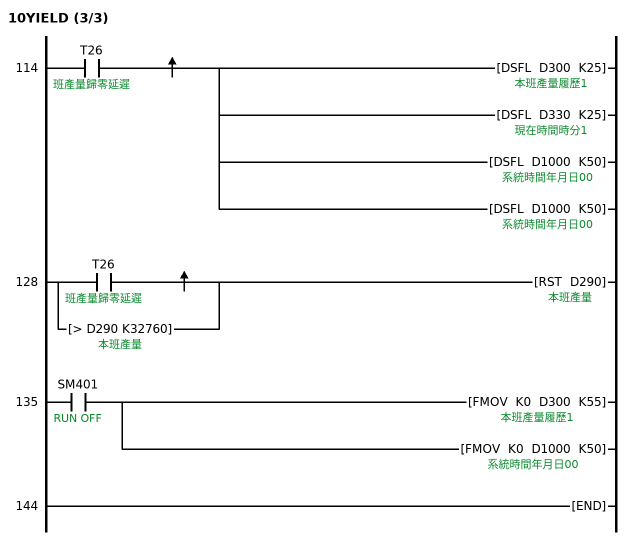
[picture p48: ladder of 10YIELD, rungs at steps 114 to 144]
114   LD      T26  ; 班產量歸零延遲
      MEP
      DSFL    D300 K25
      DSFL    D330 K25
      DSFL    D1000 K50
      DSFL    D1000 K50
128   LD      T26  ; 班產量歸零延遲
      MEP
      OR>     D290 K32760  ; 本班產量
      RST     D290  ; 本班產量
135   LD      SM401  ; RUN OFF
      FMOV    K0 D300 K55
      FMOV    K0 D1000 K50
144   END
END_PROGRAM

PROGRAM 11MAINTE
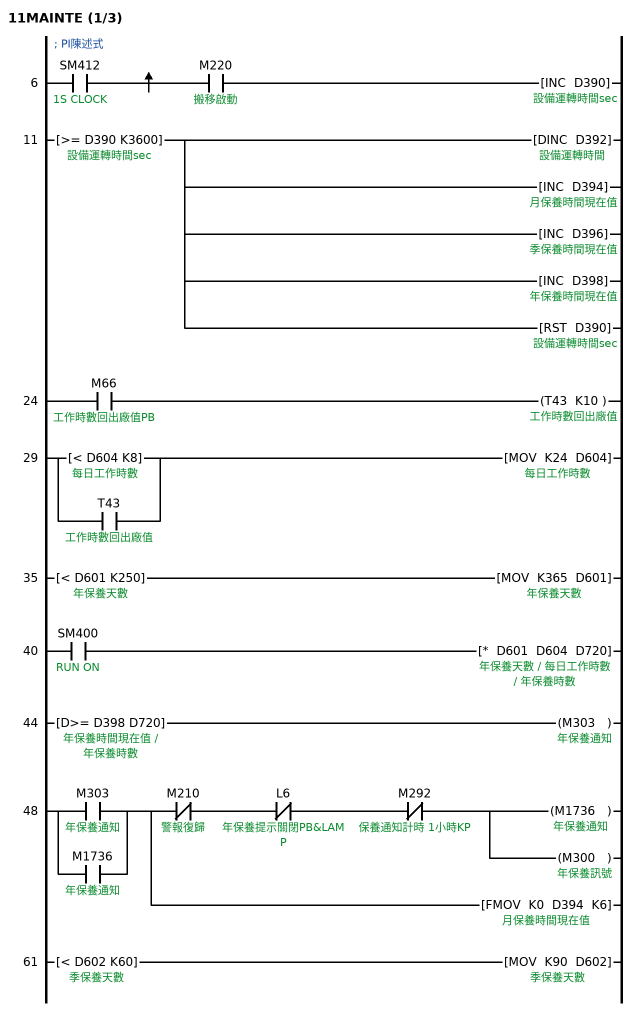
; PI陳述式
6     LD      SM412  ; 1S CLOCK
      MEP
      AND     M220  ; 搬移啟動
      INC     D390  ; 設備運轉時間sec
11    LD>=    D390 K3600  ; 設備運轉時間sec
      DINC    D392  ; 設備運轉時間
      INC     D394  ; 月保養時間現在值
      INC     D396  ; 季保養時間現在值
      INC     D398  ; 年保養時間現在值
      RST     D390  ; 設備運轉時間sec
24    LD      M66  ; 工作時數回出廠值PB
      OUT     T43 K10  ; 工作時數回出廠值
29    LD<     D604 K8  ; 每日工作時數
      OR      T43  ; 工作時數回出廠值
      MOV     K24 D604
35    LD<     D601 K250  ; 年保養天數
      MOV     K365 D601
40    LD      SM400  ; RUN ON
      *       D601 D604 D720  ; 年保養時數
44    LDD>=   D398 D720  ; 年保養時間現在值 / 年保養時數
      OUT     M303  ; 年保養通知
48    LD      M303  ; 年保養通知
      OR      M1736  ; 年保養通知
      MPS
      ANI     M210  ; 警報復歸
      ANI     L6  ; 年保養提示關閉PB&LAMP
      ANI     M292  ; 保養通知計時 1小時KP
      OUT     M1736  ; 年保養通知
      OUT     M300  ; 年保養訊號
      MPP
      FMOV    K0 D394 K6
61    LD<     D602 K60  ; 季保養天數
      MOV     K90 D602
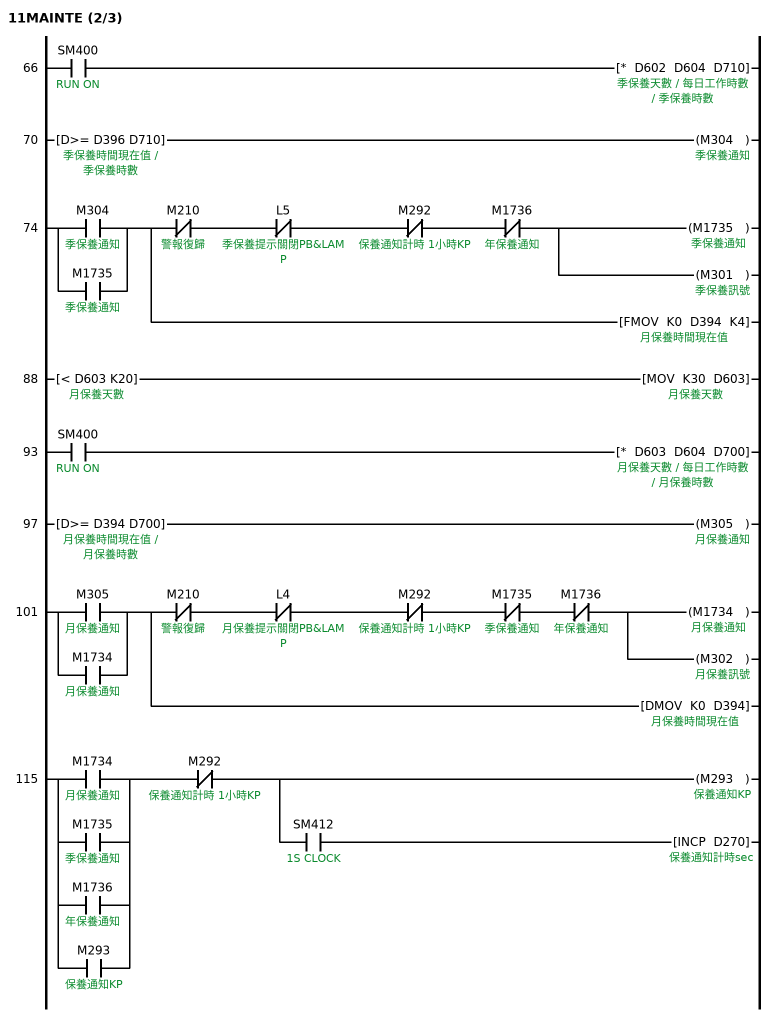
66    LD      SM400  ; RUN ON
      *       D602 D604 D710  ; 季保養時數
70    LDD>=   D396 D710  ; 季保養時間現在值 / 季保養時數
      OUT     M304  ; 季保養通知
74    LD      M304  ; 季保養通知
      OR      M1735  ; 季保養通知
      MPS
      ANI     M210  ; 警報復歸
      ANI     L5  ; 季保養提示關閉PB&LAMP
      ANI     M292  ; 保養通知計時 1小時KP
      ANI     M1736  ; 年保養通知
      OUT     M1735  ; 季保養通知
      OUT     M301  ; 季保養訊號
      MPP
      FMOV    K0 D394 K4
88    LD<     D603 K20  ; 月保養天數
      MOV     K30 D603
93    LD      SM400  ; RUN ON
      *       D603 D604 D700  ; 月保養時數
97    LDD>=   D394 D700  ; 月保養時間現在值 / 月保養時數
      OUT     M305  ; 月保養通知
101   LD      M305  ; 月保養通知
      OR      M1734  ; 月保養通知
      MPS
      ANI     M210  ; 警報復歸
      ANI     L4  ; 月保養提示關閉PB&LAMP
      ANI     M292  ; 保養通知計時 1小時KP
      ANI     M1735  ; 季保養通知
      ANI     M1736  ; 年保養通知
      OUT     M1734  ; 月保養通知
      OUT     M302  ; 月保養訊號
      MPP
      DMOV    K0 D394
115   LD      M1734  ; 月保養通知
      OR      M1735  ; 季保養通知
      OR      M1736  ; 年保養通知
      OR      M293  ; 保養通知KP
      ANI     M292  ; 保養通知計時 1小時KP
      OUT     M293  ; 保養通知KP
      AND     SM412  ; 1S CLOCK
      INCP    D270  ; 保養通知計時sec
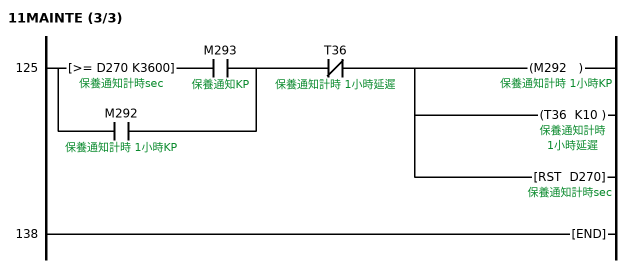
125   LD>=    D270 K3600  ; 保養通知計時sec
      AND     M293  ; 保養通知KP
      OR      M292  ; 保養通知計時 1小時KP
      ANI     T36  ; 保養通知計時 1小時延遲
      OUT     M292  ; 保養通知計時 1小時KP
      OUT     T36 K10  ; 保養通知計時 1小時延遲
      RST     D270  ; 保養通知計時sec
138   END
END_PROGRAM

PROGRAM 12ALARM1
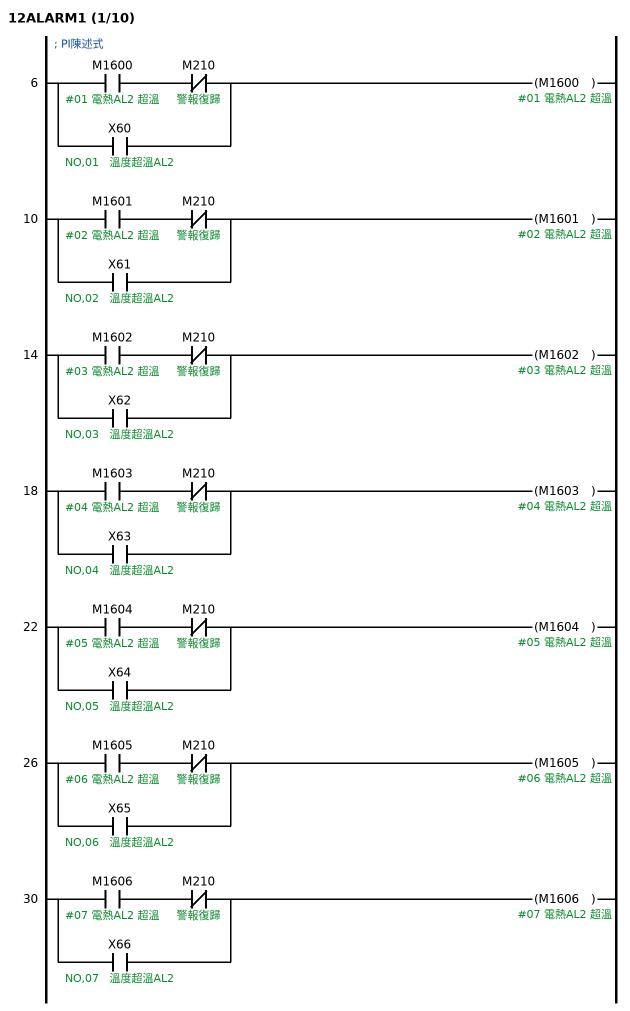
; PI陳述式
6     LD      M1600  ; #01 電熱AL2 超溫
      ANI     M210  ; 警報復歸
      OR      X60  ; NO,01   溫度超溫AL2
      OUT     M1600  ; #01 電熱AL2 超溫
10    LD      M1601  ; #02 電熱AL2 超溫
      ANI     M210  ; 警報復歸
      OR      X61  ; NO,02   溫度超溫AL2
      OUT     M1601  ; #02 電熱AL2 超溫
14    LD      M1602  ; #03 電熱AL2 超溫
      ANI     M210  ; 警報復歸
      OR      X62  ; NO,03   溫度超溫AL2
      OUT     M1602  ; #03 電熱AL2 超溫
18    LD      M1603  ; #04 電熱AL2 超溫
      ANI     M210  ; 警報復歸
      OR      X63  ; NO,04   溫度超溫AL2
      OUT     M1603  ; #04 電熱AL2 超溫
22    LD      M1604  ; #05 電熱AL2 超溫
      ANI     M210  ; 警報復歸
      OR      X64  ; NO,05   溫度超溫AL2
      OUT     M1604  ; #05 電熱AL2 超溫
26    LD      M1605  ; #06 電熱AL2 超溫
      ANI     M210  ; 警報復歸
      OR      X65  ; NO,06   溫度超溫AL2
      OUT     M1605  ; #06 電熱AL2 超溫
30    LD      M1606  ; #07 電熱AL2 超溫
      ANI     M210  ; 警報復歸
      OR      X66  ; NO,07   溫度超溫AL2
      OUT     M1606  ; #07 電熱AL2 超溫
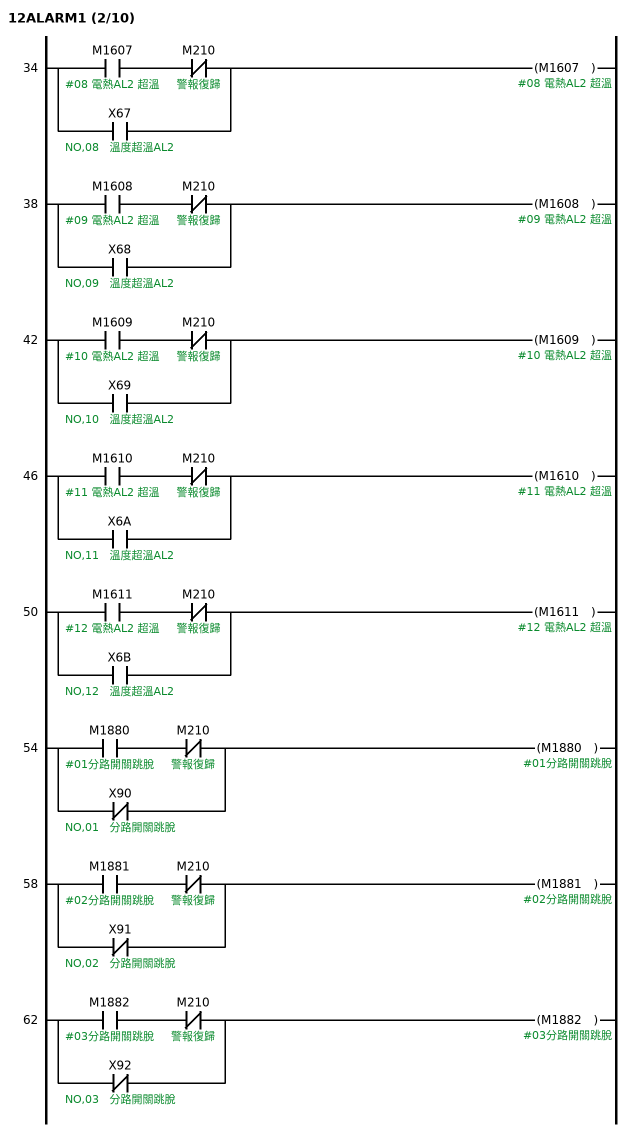
34    LD      M1607  ; #08 電熱AL2 超溫
      ANI     M210  ; 警報復歸
      OR      X67  ; NO,08   溫度超溫AL2
      OUT     M1607  ; #08 電熱AL2 超溫
38    LD      M1608  ; #09 電熱AL2 超溫
      ANI     M210  ; 警報復歸
      OR      X68  ; NO,09   溫度超溫AL2
      OUT     M1608  ; #09 電熱AL2 超溫
42    LD      M1609  ; #10 電熱AL2 超溫
      ANI     M210  ; 警報復歸
      OR      X69  ; NO,10   溫度超溫AL2
      OUT     M1609  ; #10 電熱AL2 超溫
46    LD      M1610  ; #11 電熱AL2 超溫
      ANI     M210  ; 警報復歸
      OR      X6A  ; NO,11   溫度超溫AL2
      OUT     M1610  ; #11 電熱AL2 超溫
50    LD      M1611  ; #12 電熱AL2 超溫
      ANI     M210  ; 警報復歸
      OR      X6B  ; NO,12   溫度超溫AL2
      OUT     M1611  ; #12 電熱AL2 超溫
54    LD      M1880  ; #01分路開關跳脫
      ANI     M210  ; 警報復歸
      ORI     X90  ; NO,01   分路開關跳脫
      OUT     M1880  ; #01分路開關跳脫
58    LD      M1881  ; #02分路開關跳脫
      ANI     M210  ; 警報復歸
      ORI     X91  ; NO,02   分路開關跳脫
      OUT     M1881  ; #02分路開關跳脫
62    LD      M1882  ; #03分路開關跳脫
      ANI     M210  ; 警報復歸
      ORI     X92  ; NO,03   分路開關跳脫
      OUT     M1882  ; #03分路開關跳脫
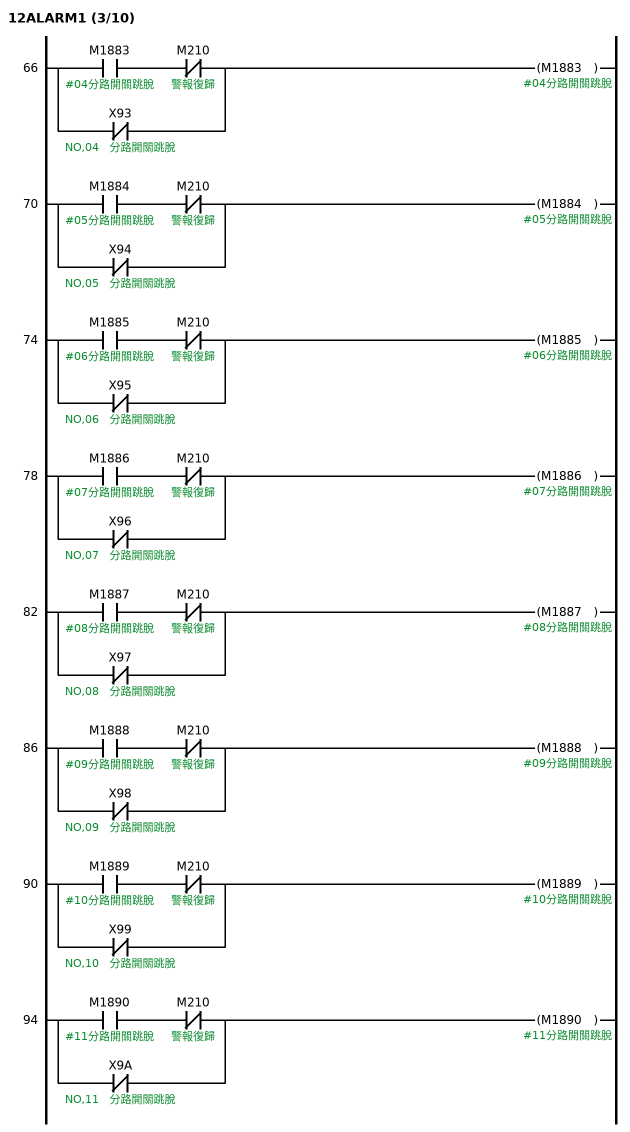
66    LD      M1883  ; #04分路開關跳脫
      ANI     M210  ; 警報復歸
      ORI     X93  ; NO,04   分路開關跳脫
      OUT     M1883  ; #04分路開關跳脫
70    LD      M1884  ; #05分路開關跳脫
      ANI     M210  ; 警報復歸
      ORI     X94  ; NO,05   分路開關跳脫
      OUT     M1884  ; #05分路開關跳脫
74    LD      M1885  ; #06分路開關跳脫
      ANI     M210  ; 警報復歸
      ORI     X95  ; NO,06   分路開關跳脫
      OUT     M1885  ; #06分路開關跳脫
78    LD      M1886  ; #07分路開關跳脫
      ANI     M210  ; 警報復歸
      ORI     X96  ; NO,07   分路開關跳脫
      OUT     M1886  ; #07分路開關跳脫
82    LD      M1887  ; #08分路開關跳脫
      ANI     M210  ; 警報復歸
      ORI     X97  ; NO,08   分路開關跳脫
      OUT     M1887  ; #08分路開關跳脫
86    LD      M1888  ; #09分路開關跳脫
      ANI     M210  ; 警報復歸
      ORI     X98  ; NO,09   分路開關跳脫
      OUT     M1888  ; #09分路開關跳脫
90    LD      M1889  ; #10分路開關跳脫
      ANI     M210  ; 警報復歸
      ORI     X99  ; NO,10   分路開關跳脫
      OUT     M1889  ; #10分路開關跳脫
94    LD      M1890  ; #11分路開關跳脫
      ANI     M210  ; 警報復歸
      ORI     X9A  ; NO,11   分路開關跳脫
      OUT     M1890  ; #11分路開關跳脫
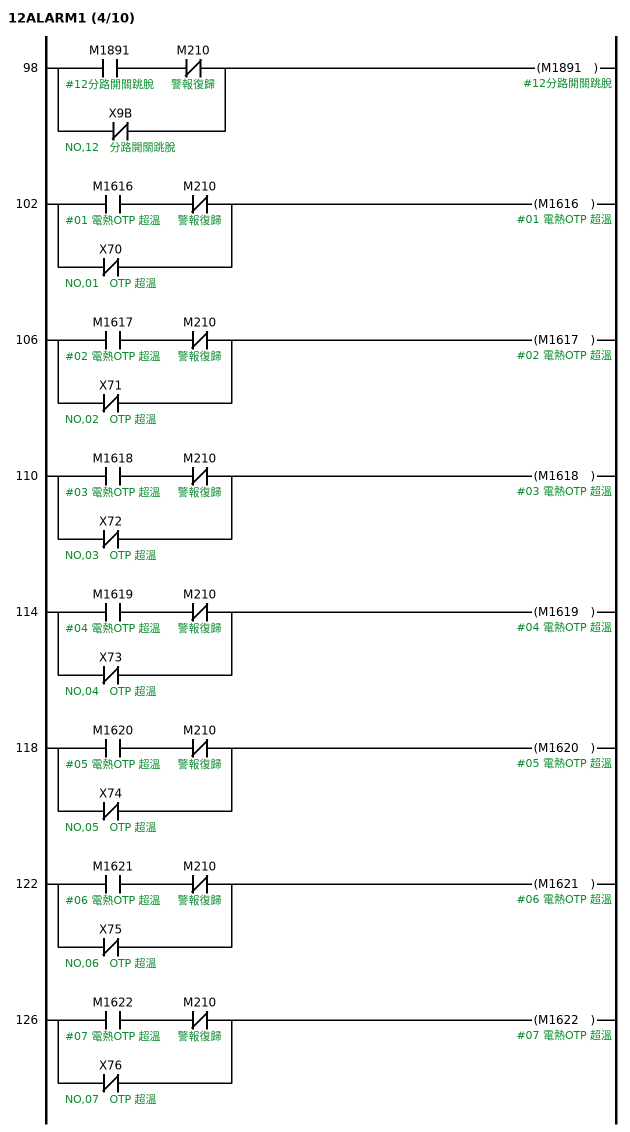
98    LD      M1891  ; #12分路開關跳脫
      ANI     M210  ; 警報復歸
      ORI     X9B  ; NO,12   分路開關跳脫
      OUT     M1891  ; #12分路開關跳脫
102   LD      M1616  ; #01 電熱OTP 超溫
      ANI     M210  ; 警報復歸
      ORI     X70  ; NO,01   OTP 超溫
      OUT     M1616  ; #01 電熱OTP 超溫
106   LD      M1617  ; #02 電熱OTP 超溫
      ANI     M210  ; 警報復歸
      ORI     X71  ; NO,02   OTP 超溫
      OUT     M1617  ; #02 電熱OTP 超溫
110   LD      M1618  ; #03 電熱OTP 超溫
      ANI     M210  ; 警報復歸
      ORI     X72  ; NO,03   OTP 超溫
      OUT     M1618  ; #03 電熱OTP 超溫
114   LD      M1619  ; #04 電熱OTP 超溫
      ANI     M210  ; 警報復歸
      ORI     X73  ; NO,04   OTP 超溫
      OUT     M1619  ; #04 電熱OTP 超溫
118   LD      M1620  ; #05 電熱OTP 超溫
      ANI     M210  ; 警報復歸
      ORI     X74  ; NO,05   OTP 超溫
      OUT     M1620  ; #05 電熱OTP 超溫
122   LD      M1621  ; #06 電熱OTP 超溫
      ANI     M210  ; 警報復歸
      ORI     X75  ; NO,06   OTP 超溫
      OUT     M1621  ; #06 電熱OTP 超溫
126   LD      M1622  ; #07 電熱OTP 超溫
      ANI     M210  ; 警報復歸
      ORI     X76  ; NO,07   OTP 超溫
      OUT     M1622  ; #07 電熱OTP 超溫
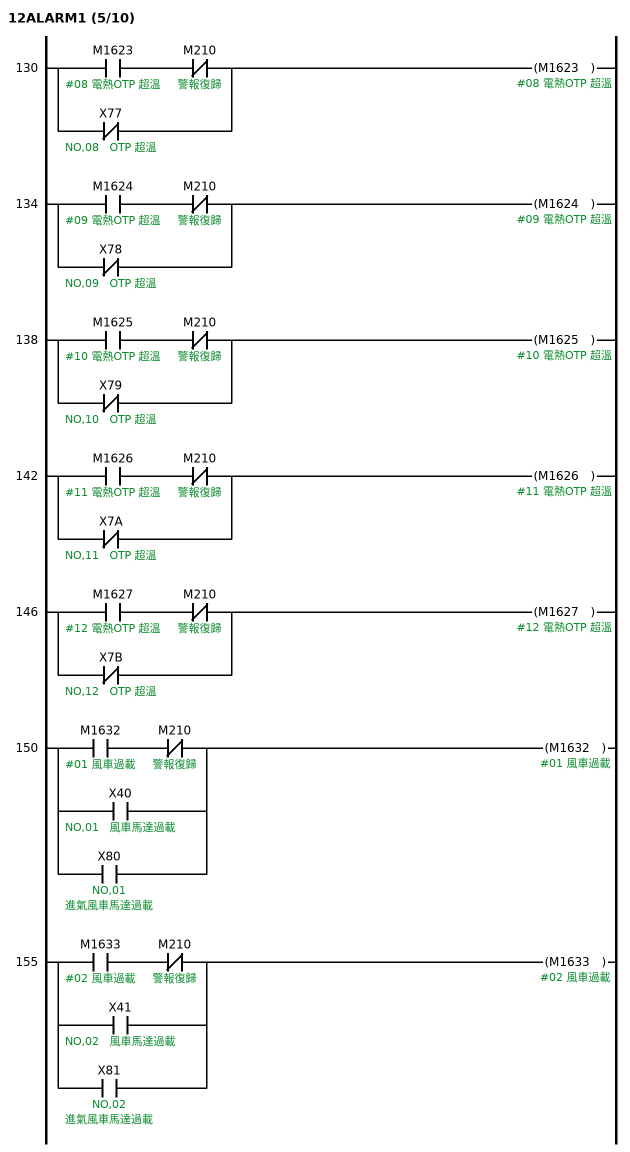
130   LD      M1623  ; #08 電熱OTP 超溫
      ANI     M210  ; 警報復歸
      ORI     X77  ; NO,08   OTP 超溫
      OUT     M1623  ; #08 電熱OTP 超溫
134   LD      M1624  ; #09 電熱OTP 超溫
      ANI     M210  ; 警報復歸
      ORI     X78  ; NO,09   OTP 超溫
      OUT     M1624  ; #09 電熱OTP 超溫
138   LD      M1625  ; #10 電熱OTP 超溫
      ANI     M210  ; 警報復歸
      ORI     X79  ; NO,10   OTP 超溫
      OUT     M1625  ; #10 電熱OTP 超溫
142   LD      M1626  ; #11 電熱OTP 超溫
      ANI     M210  ; 警報復歸
      ORI     X7A  ; NO,11   OTP 超溫
      OUT     M1626  ; #11 電熱OTP 超溫
146   LD      M1627  ; #12 電熱OTP 超溫
      ANI     M210  ; 警報復歸
      ORI     X7B  ; NO,12   OTP 超溫
      OUT     M1627  ; #12 電熱OTP 超溫
150   LD      M1632  ; #01 風車過載
      ANI     M210  ; 警報復歸
      OR      X40  ; NO,01   風車馬達過載
      OR      X80  ; NO,01   進氣風車馬達過載
      OUT     M1632  ; #01 風車過載
155   LD      M1633  ; #02 風車過載
      ANI     M210  ; 警報復歸
      OR      X41  ; NO,02   風車馬達過載
      OR      X81  ; NO,02   進氣風車馬達過載
      OUT     M1633  ; #02 風車過載
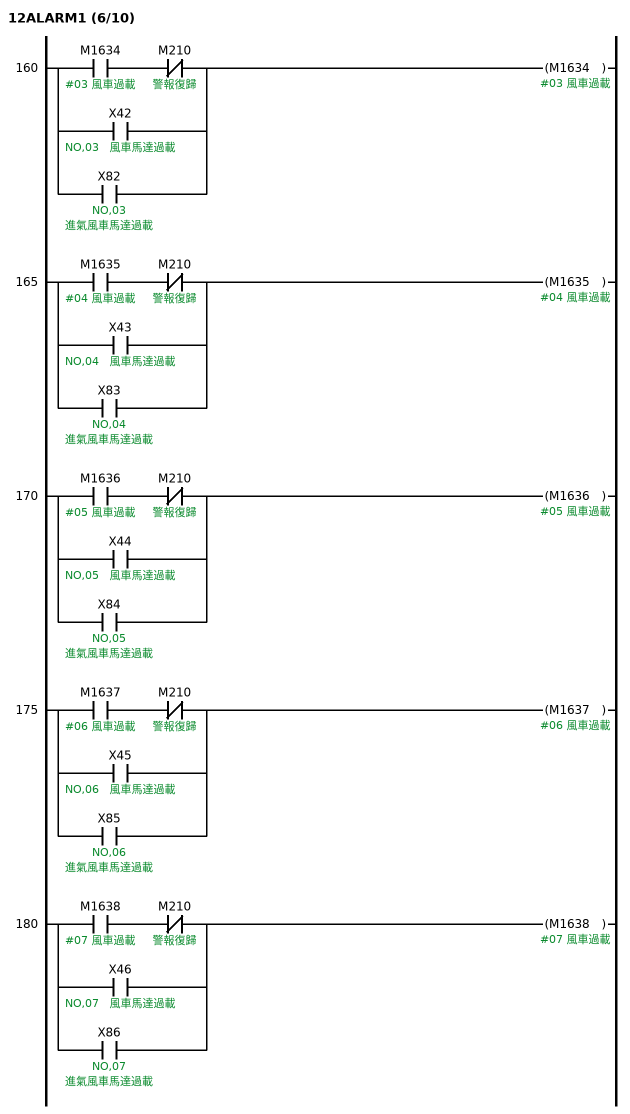
160   LD      M1634  ; #03 風車過載
      ANI     M210  ; 警報復歸
      OR      X42  ; NO,03   風車馬達過載
      OR      X82  ; NO,03   進氣風車馬達過載
      OUT     M1634  ; #03 風車過載
165   LD      M1635  ; #04 風車過載
      ANI     M210  ; 警報復歸
      OR      X43  ; NO,04   風車馬達過載
      OR      X83  ; NO,04   進氣風車馬達過載
      OUT     M1635  ; #04 風車過載
170   LD      M1636  ; #05 風車過載
      ANI     M210  ; 警報復歸
      OR      X44  ; NO,05   風車馬達過載
      OR      X84  ; NO,05   進氣風車馬達過載
      OUT     M1636  ; #05 風車過載
175   LD      M1637  ; #06 風車過載
      ANI     M210  ; 警報復歸
      OR      X45  ; NO,06   風車馬達過載
      OR      X85  ; NO,06   進氣風車馬達過載
      OUT     M1637  ; #06 風車過載
180   LD      M1638  ; #07 風車過載
      ANI     M210  ; 警報復歸
      OR      X46  ; NO,07   風車馬達過載
      OR      X86  ; NO,07   進氣風車馬達過載
      OUT     M1638  ; #07 風車過載
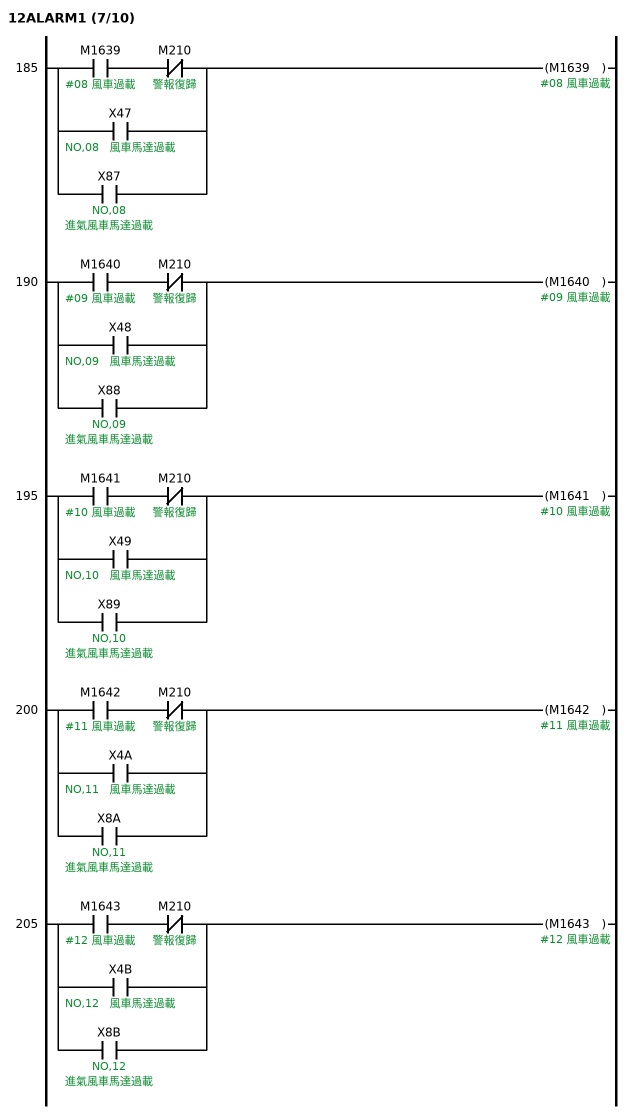
185   LD      M1639  ; #08 風車過載
      ANI     M210  ; 警報復歸
      OR      X47  ; NO,08   風車馬達過載
      OR      X87  ; NO,08   進氣風車馬達過載
      OUT     M1639  ; #08 風車過載
190   LD      M1640  ; #09 風車過載
      ANI     M210  ; 警報復歸
      OR      X48  ; NO,09   風車馬達過載
      OR      X88  ; NO,09   進氣風車馬達過載
      OUT     M1640  ; #09 風車過載
195   LD      M1641  ; #10 風車過載
      ANI     M210  ; 警報復歸
      OR      X49  ; NO,10   風車馬達過載
      OR      X89  ; NO,10   進氣風車馬達過載
      OUT     M1641  ; #10 風車過載
200   LD      M1642  ; #11 風車過載
      ANI     M210  ; 警報復歸
      OR      X4A  ; NO,11   風車馬達過載
      OR      X8A  ; NO,11   進氣風車馬達過載
      OUT     M1642  ; #11 風車過載
205   LD      M1643  ; #12 風車過載
      ANI     M210  ; 警報復歸
      OR      X4B  ; NO,12   風車馬達過載
      OR      X8B  ; NO,12   進氣風車馬達過載
      OUT     M1643  ; #12 風車過載
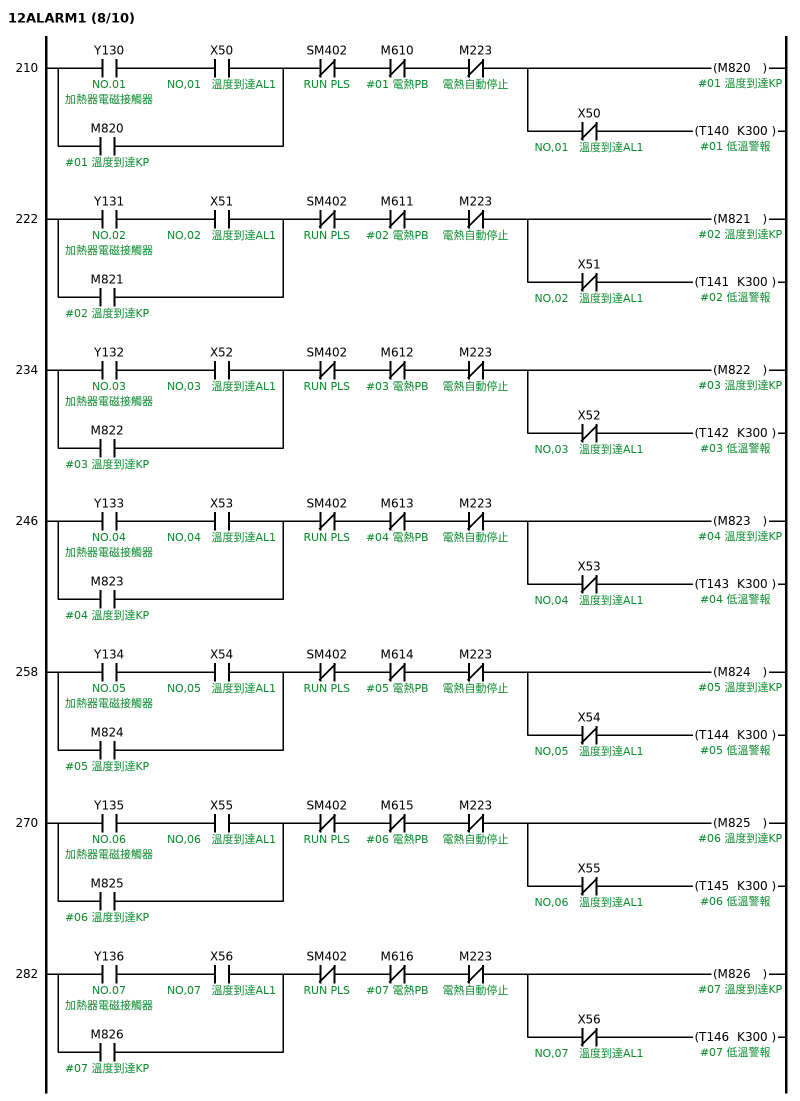
210   LD      Y130  ; NO.01   加熱器電磁接觸器
      AND     X50  ; NO,01   溫度到達AL1
      OR      M820  ; #01 溫度到達KP
      ANI     SM402  ; RUN PLS
      ANI     M610  ; #01 電熱PB
      ANI     M223  ; 電熱自動停止
      OUT     M820  ; #01 溫度到達KP
      ANI     X50  ; NO,01   溫度到達AL1
      OUT     T140 K300  ; #01 低溫警報
222   LD      Y131  ; NO.02   加熱器電磁接觸器
      AND     X51  ; NO,02   溫度到達AL1
      OR      M821  ; #02 溫度到達KP
      ANI     SM402  ; RUN PLS
      ANI     M611  ; #02 電熱PB
      ANI     M223  ; 電熱自動停止
      OUT     M821  ; #02 溫度到達KP
      ANI     X51  ; NO,02   溫度到達AL1
      OUT     T141 K300  ; #02 低溫警報
234   LD      Y132  ; NO.03   加熱器電磁接觸器
      AND     X52  ; NO,03   溫度到達AL1
      OR      M822  ; #03 溫度到達KP
      ANI     SM402  ; RUN PLS
      ANI     M612  ; #03 電熱PB
      ANI     M223  ; 電熱自動停止
      OUT     M822  ; #03 溫度到達KP
      ANI     X52  ; NO,03   溫度到達AL1
      OUT     T142 K300  ; #03 低溫警報
246   LD      Y133  ; NO.04   加熱器電磁接觸器
      AND     X53  ; NO,04   溫度到達AL1
      OR      M823  ; #04 溫度到達KP
      ANI     SM402  ; RUN PLS
      ANI     M613  ; #04 電熱PB
      ANI     M223  ; 電熱自動停止
      OUT     M823  ; #04 溫度到達KP
      ANI     X53  ; NO,04   溫度到達AL1
      OUT     T143 K300  ; #04 低溫警報
258   LD      Y134  ; NO.05   加熱器電磁接觸器
      AND     X54  ; NO,05   溫度到達AL1
      OR      M824  ; #05 溫度到達KP
      ANI     SM402  ; RUN PLS
      ANI     M614  ; #05 電熱PB
      ANI     M223  ; 電熱自動停止
      OUT     M824  ; #05 溫度到達KP
      ANI     X54  ; NO,05   溫度到達AL1
      OUT     T144 K300  ; #05 低溫警報
270   LD      Y135  ; NO.06   加熱器電磁接觸器
      AND     X55  ; NO,06   溫度到達AL1
      OR      M825  ; #06 溫度到達KP
      ANI     SM402  ; RUN PLS
      ANI     M615  ; #06 電熱PB
      ANI     M223  ; 電熱自動停止
      OUT     M825  ; #06 溫度到達KP
      ANI     X55  ; NO,06   溫度到達AL1
      OUT     T145 K300  ; #06 低溫警報
282   LD      Y136  ; NO.07   加熱器電磁接觸器
      AND     X56  ; NO,07   溫度到達AL1
      OR      M826  ; #07 溫度到達KP
      ANI     SM402  ; RUN PLS
      ANI     M616  ; #07 電熱PB
      ANI     M223  ; 電熱自動停止
      OUT     M826  ; #07 溫度到達KP
      ANI     X56  ; NO,07   溫度到達AL1
      OUT     T146 K300  ; #07 低溫警報
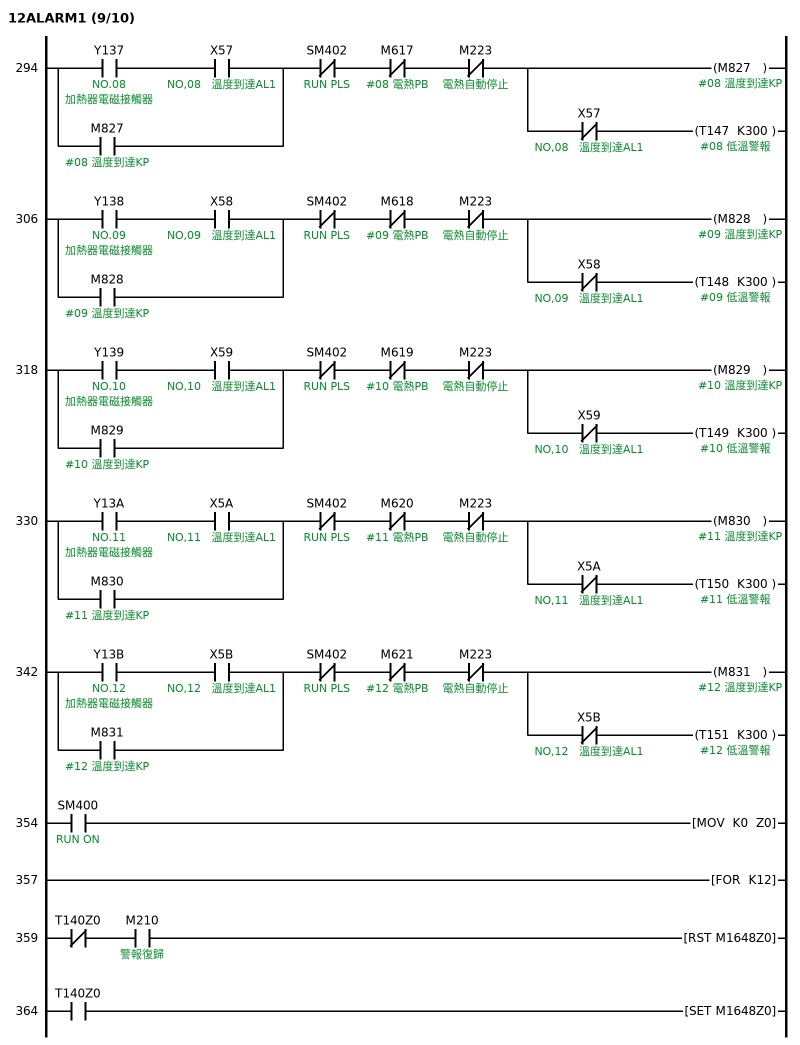
294   LD      Y137  ; NO.08   加熱器電磁接觸器
      AND     X57  ; NO,08   溫度到達AL1
      OR      M827  ; #08 溫度到達KP
      ANI     SM402  ; RUN PLS
      ANI     M617  ; #08 電熱PB
      ANI     M223  ; 電熱自動停止
      OUT     M827  ; #08 溫度到達KP
      ANI     X57  ; NO,08   溫度到達AL1
      OUT     T147 K300  ; #08 低溫警報
306   LD      Y138  ; NO.09   加熱器電磁接觸器
      AND     X58  ; NO,09   溫度到達AL1
      OR      M828  ; #09 溫度到達KP
      ANI     SM402  ; RUN PLS
      ANI     M618  ; #09 電熱PB
      ANI     M223  ; 電熱自動停止
      OUT     M828  ; #09 溫度到達KP
      ANI     X58  ; NO,09   溫度到達AL1
      OUT     T148 K300  ; #09 低溫警報
318   LD      Y139  ; NO.10   加熱器電磁接觸器
      AND     X59  ; NO,10   溫度到達AL1
      OR      M829  ; #10 溫度到達KP
      ANI     SM402  ; RUN PLS
      ANI     M619  ; #10 電熱PB
      ANI     M223  ; 電熱自動停止
      OUT     M829  ; #10 溫度到達KP
      ANI     X59  ; NO,10   溫度到達AL1
      OUT     T149 K300  ; #10 低溫警報
330   LD      Y13A  ; NO.11   加熱器電磁接觸器
      AND     X5A  ; NO,11   溫度到達AL1
      OR      M830  ; #11 溫度到達KP
      ANI     SM402  ; RUN PLS
      ANI     M620  ; #11 電熱PB
      ANI     M223  ; 電熱自動停止
      OUT     M830  ; #11 溫度到達KP
      ANI     X5A  ; NO,11   溫度到達AL1
      OUT     T150 K300  ; #11 低溫警報
342   LD      Y13B  ; NO.12   加熱器電磁接觸器
      AND     X5B  ; NO,12   溫度到達AL1
      OR      M831  ; #12 溫度到達KP
      ANI     SM402  ; RUN PLS
      ANI     M621  ; #12 電熱PB
      ANI     M223  ; 電熱自動停止
      OUT     M831  ; #12 溫度到達KP
      ANI     X5B  ; NO,12   溫度到達AL1
      OUT     T151 K300  ; #12 低溫警報
354   LD      SM400  ; RUN ON
      MOV     K0 Z0
357   FOR     K12
359   LDI     T140Z0
      AND     M210  ; 警報復歸
      RST     M1648Z0
364   LD      T140Z0
      SET     M1648Z0
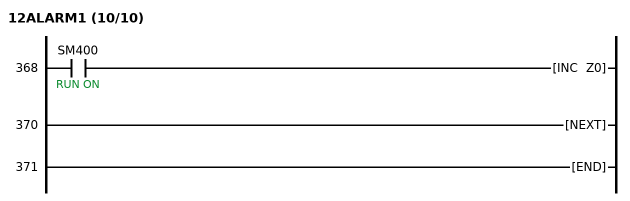
368   LD      SM400  ; RUN ON
      INC     Z0
370   NEXT
371   END
END_PROGRAM

PROGRAM 13ALARM2
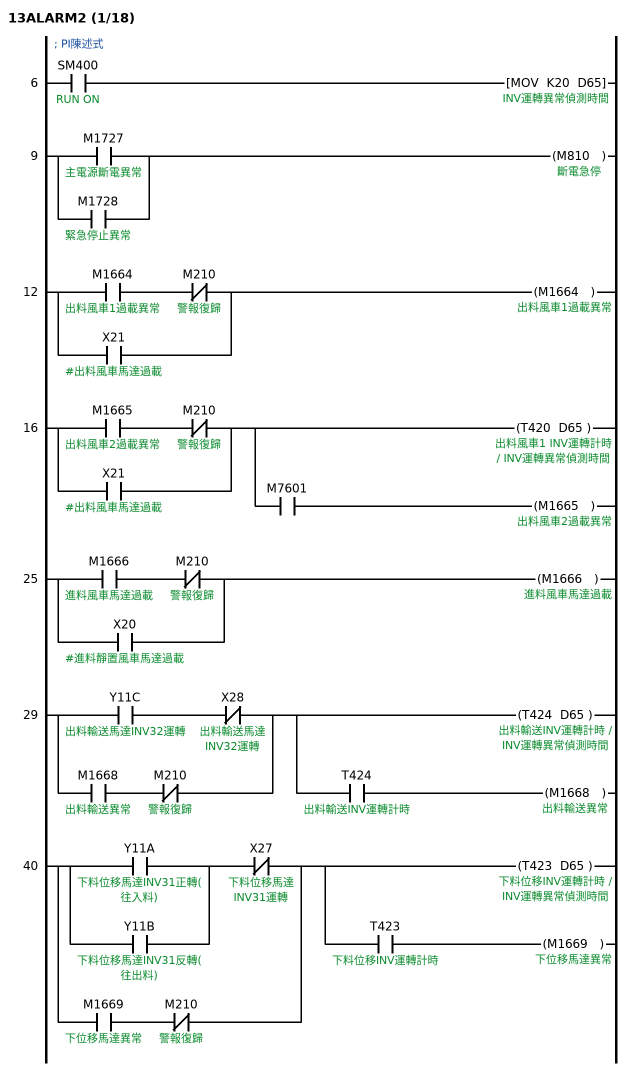
; PI陳述式
6     LD      SM400  ; RUN ON
      MOV     K20 D65  ; INV運轉異常偵測時間
9     LD      M1727  ; 主電源斷電異常
      OR      M1728  ; 緊急停止異常
      OUT     M810  ; 斷電急停
12    LD      M1664  ; 出料風車1過載異常
      ANI     M210  ; 警報復歸
      OR      X21  ; #出料風車馬達過載
      OUT     M1664  ; 出料風車1過載異常
16    LD      M1665  ; 出料風車2過載異常
      ANI     M210  ; 警報復歸
      OR      X21  ; #出料風車馬達過載
      OUT     T420 D65  ; 出料風車1 INV運轉計時 / INV運轉異常偵測時間
      AND     M7601
      OUT     M1665  ; 出料風車2過載異常
25    LD      M1666  ; 進料風車馬達過載
      ANI     M210  ; 警報復歸
      OR      X20  ; #進料靜置風車馬達過載
      OUT     M1666  ; 進料風車馬達過載
29    LD      Y11C  ; 出料輸送馬達INV32運轉
      ANI     X28  ; 出料輸送馬達    INV32運轉
      LD      M1668  ; 出料輸送異常
      ANI     M210  ; 警報復歸
      ORB
      OUT     T424 D65  ; 出料輸送INV運轉計時 / INV運轉異常偵測時間
      AND     T424  ; 出料輸送INV運轉計時
      OUT     M1668  ; 出料輸送異常
40    LD      Y11A  ; 下料位移馬達INV31正轉(往入料)
      OR      Y11B  ; 下料位移馬達INV31反轉(往出料)
      ANI     X27  ; 下料位移馬達    INV31運轉
      LD      M1669  ; 下位移馬達異常
      ANI     M210  ; 警報復歸
      ORB
      OUT     T423 D65  ; 下料位移INV運轉計時 / INV運轉異常偵測時間
      AND     T423  ; 下料位移INV運轉計時
      OUT     M1669  ; 下位移馬達異常
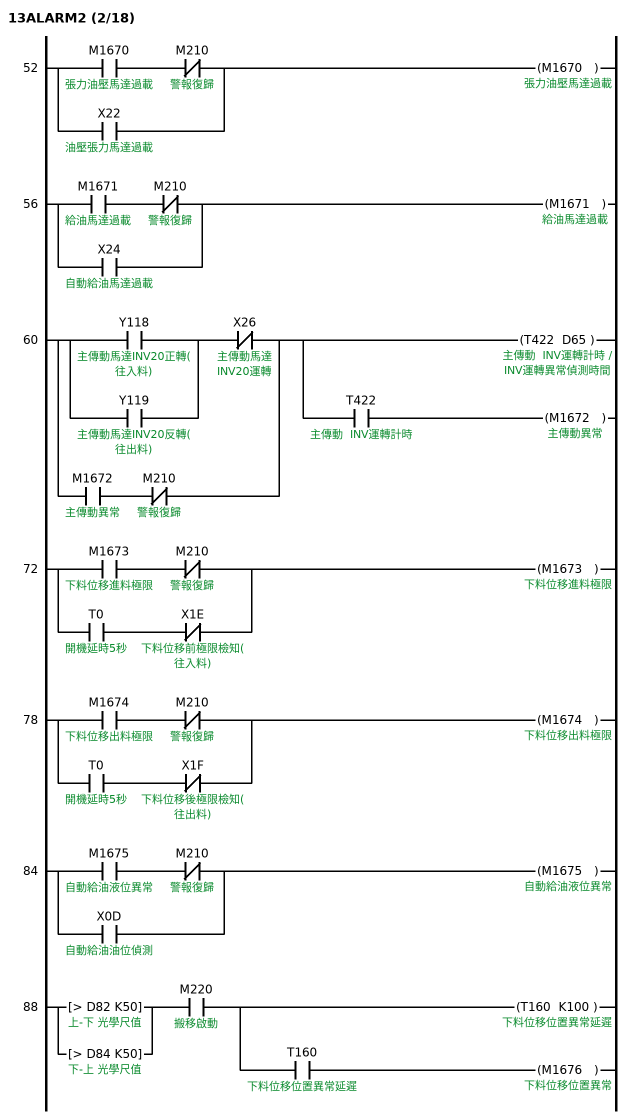
52    LD      M1670  ; 張力油壓馬達過載
      ANI     M210  ; 警報復歸
      OR      X22  ; 油壓張力馬達過載
      OUT     M1670  ; 張力油壓馬達過載
56    LD      M1671  ; 給油馬達過載
      ANI     M210  ; 警報復歸
      OR      X24  ; 自動給油馬達過載
      OUT     M1671  ; 給油馬達過載
60    LD      Y118  ; 主傳動馬達INV20正轉(往入料)
      OR      Y119  ; 主傳動馬達INV20反轉(往出料)
      ANI     X26  ; 主傳動馬達      INV20運轉
      LD      M1672  ; 主傳動異常
      ANI     M210  ; 警報復歸
      ORB
      OUT     T422 D65  ; 主傳動  INV運轉計時 / INV運轉異常偵測時間
      AND     T422  ; 主傳動  INV運轉計時
      OUT     M1672  ; 主傳動異常
72    LD      M1673  ; 下料位移進料極限
      ANI     M210  ; 警報復歸
      LD      T0  ; 開機延時5秒
      ANI     X1E  ; 下料位移前極限檢知(往入料)
      ORB
      OUT     M1673  ; 下料位移進料極限
78    LD      M1674  ; 下料位移出料極限
      ANI     M210  ; 警報復歸
      LD      T0  ; 開機延時5秒
      ANI     X1F  ; 下料位移後極限檢知(往出料)
      ORB
      OUT     M1674  ; 下料位移出料極限
84    LD      M1675  ; 自動給油液位異常
      ANI     M210  ; 警報復歸
      OR      X0D  ; 自動給油油位偵測
      OUT     M1675  ; 自動給油液位異常
88    LD>     D82 K50  ; 上-下 光學尺值
      OR>     D84 K50  ; 下-上 光學尺值
      AND     M220  ; 搬移啟動
      OUT     T160 K100  ; 下料位移位置異常延遲
      AND     T160  ; 下料位移位置異常延遲
      OUT     M1676  ; 下料位移位置異常
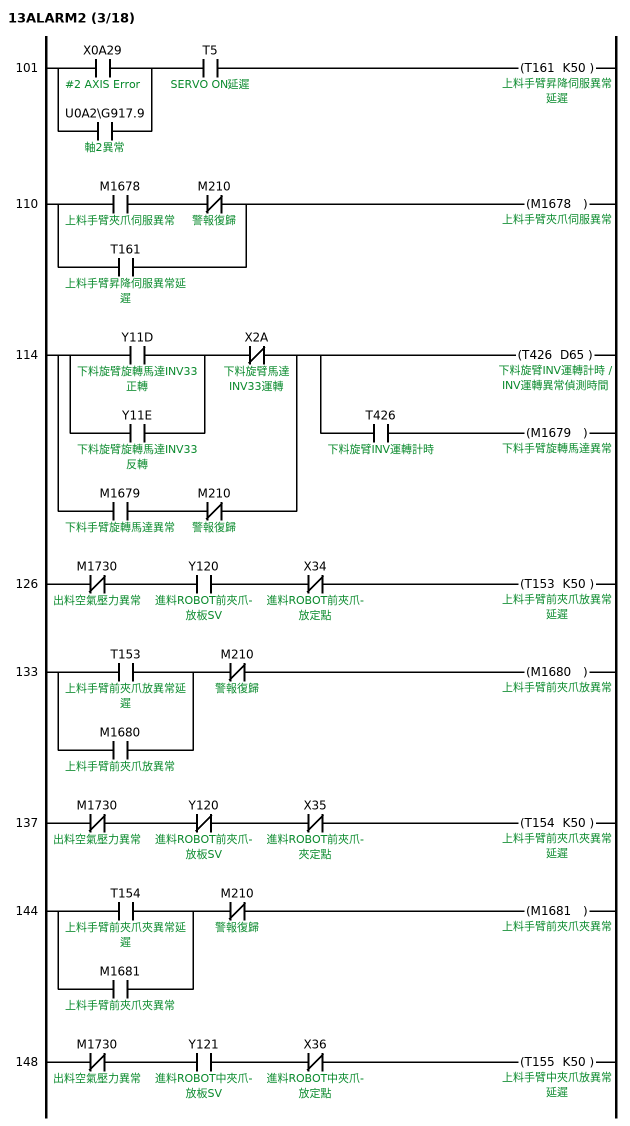
101   LD      X0A29  ; #2 AXIS Error
      OR      U0A2\G917.9  ; 軸2異常
      AND     T5  ; SERVO ON延遲
      OUT     T161 K50  ; 上料手臂昇降伺服異常延遲
110   LD      M1678  ; 上料手臂夾爪伺服異常
      ANI     M210  ; 警報復歸
      OR      T161  ; 上料手臂昇降伺服異常延遲
      OUT     M1678  ; 上料手臂夾爪伺服異常
114   LD      Y11D  ; 下料旋臂旋轉馬達INV33正轉
      OR      Y11E  ; 下料旋臂旋轉馬達INV33反轉
      ANI     X2A  ; 下料旋臂馬達    INV33運轉
      LD      M1679  ; 下料手臂旋轉馬達異常
      ANI     M210  ; 警報復歸
      ORB
      OUT     T426 D65  ; 下料旋臂INV運轉計時 / INV運轉異常偵測時間
      AND     T426  ; 下料旋臂INV運轉計時
      OUT     M1679  ; 下料手臂旋轉馬達異常
126   LDI     M1730  ; 出料空氣壓力異常
      AND     Y120  ; 進料ROBOT前夾爪-放板SV
      ANI     X34  ; 進料ROBOT前夾爪-放定點
      OUT     T153 K50  ; 上料手臂前夾爪放異常延遲
133   LD      T153  ; 上料手臂前夾爪放異常延遲
      OR      M1680  ; 上料手臂前夾爪放異常
      ANI     M210  ; 警報復歸
      OUT     M1680  ; 上料手臂前夾爪放異常
137   LDI     M1730  ; 出料空氣壓力異常
      ANI     Y120  ; 進料ROBOT前夾爪-放板SV
      ANI     X35  ; 進料ROBOT前夾爪-夾定點
      OUT     T154 K50  ; 上料手臂前夾爪夾異常延遲
144   LD      T154  ; 上料手臂前夾爪夾異常延遲
      OR      M1681  ; 上料手臂前夾爪夾異常
      ANI     M210  ; 警報復歸
      OUT     M1681  ; 上料手臂前夾爪夾異常
148   LDI     M1730  ; 出料空氣壓力異常
      AND     Y121  ; 進料ROBOT中夾爪-放板SV
      ANI     X36  ; 進料ROBOT中夾爪-放定點
      OUT     T155 K50  ; 上料手臂中夾爪放異常延遲
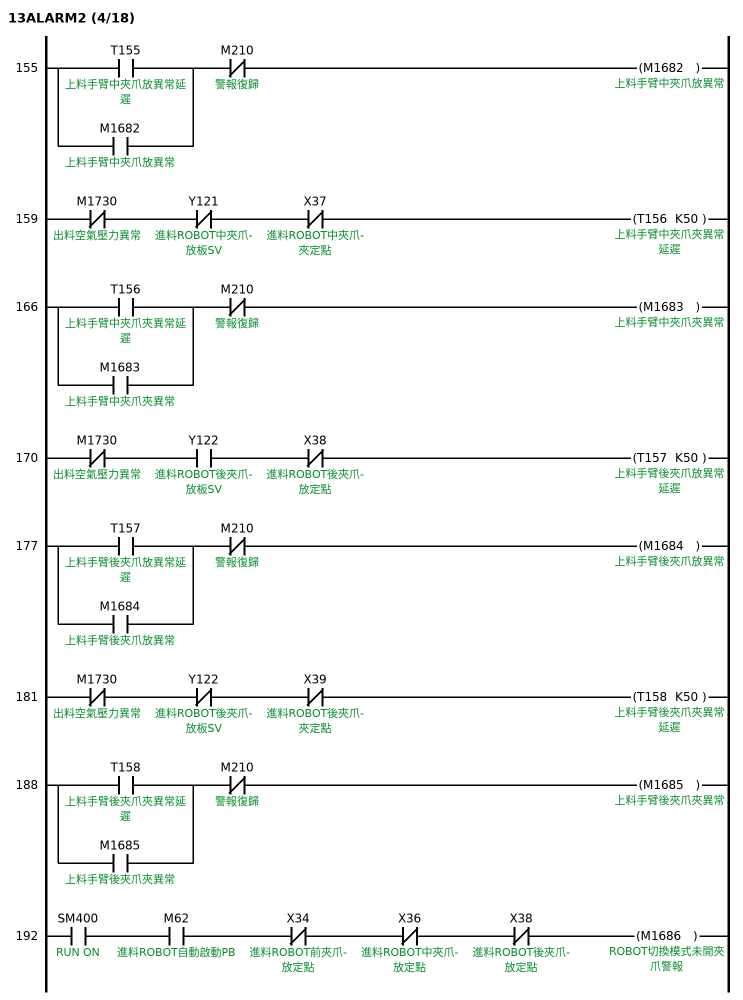
155   LD      T155  ; 上料手臂中夾爪放異常延遲
      OR      M1682  ; 上料手臂中夾爪放異常
      ANI     M210  ; 警報復歸
      OUT     M1682  ; 上料手臂中夾爪放異常
159   LDI     M1730  ; 出料空氣壓力異常
      ANI     Y121  ; 進料ROBOT中夾爪-放板SV
      ANI     X37  ; 進料ROBOT中夾爪-夾定點
      OUT     T156 K50  ; 上料手臂中夾爪夾異常延遲
166   LD      T156  ; 上料手臂中夾爪夾異常延遲
      OR      M1683  ; 上料手臂中夾爪夾異常
      ANI     M210  ; 警報復歸
      OUT     M1683  ; 上料手臂中夾爪夾異常
170   LDI     M1730  ; 出料空氣壓力異常
      AND     Y122  ; 進料ROBOT後夾爪-放板SV
      ANI     X38  ; 進料ROBOT後夾爪-放定點
      OUT     T157 K50  ; 上料手臂後夾爪放異常延遲
177   LD      T157  ; 上料手臂後夾爪放異常延遲
      OR      M1684  ; 上料手臂後夾爪放異常
      ANI     M210  ; 警報復歸
      OUT     M1684  ; 上料手臂後夾爪放異常
181   LDI     M1730  ; 出料空氣壓力異常
      ANI     Y122  ; 進料ROBOT後夾爪-放板SV
      ANI     X39  ; 進料ROBOT後夾爪-夾定點
      OUT     T158 K50  ; 上料手臂後夾爪夾異常延遲
188   LD      T158  ; 上料手臂後夾爪夾異常延遲
      OR      M1685  ; 上料手臂後夾爪夾異常
      ANI     M210  ; 警報復歸
      OUT     M1685  ; 上料手臂後夾爪夾異常
192   LD      SM400  ; RUN ON
      AND     M62  ; 進料ROBOT自動啟動PB
      ANI     X34  ; 進料ROBOT前夾爪-放定點
      ANI     X36  ; 進料ROBOT中夾爪-放定點
      ANI     X38  ; 進料ROBOT後夾爪-放定點
      OUT     M1686  ; ROBOT切換模式未開夾爪警報
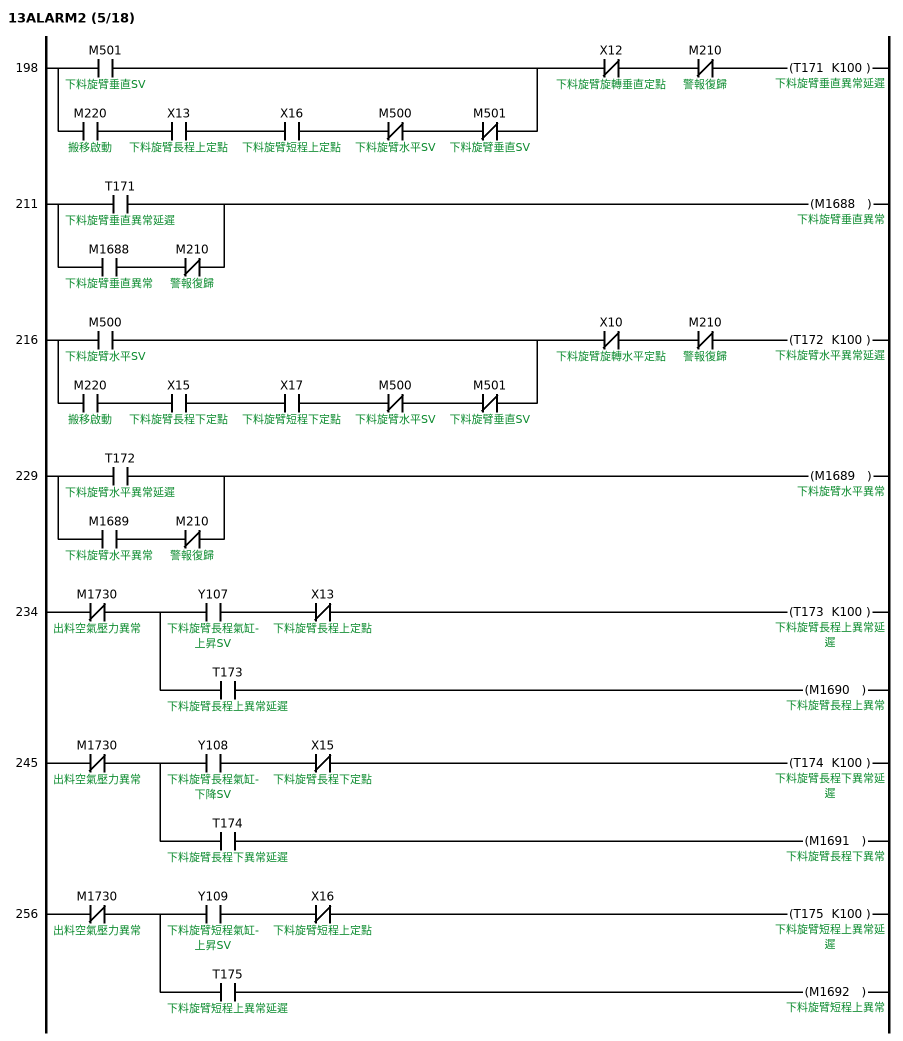
198   LD      M501  ; 下料旋臂垂直SV
      LD      M220  ; 搬移啟動
      AND     X13  ; 下料旋臂長程上定點
      AND     X16  ; 下料旋臂短程上定點
      ANI     M500  ; 下料旋臂水平SV
      ANI     M501  ; 下料旋臂垂直SV
      ORB
      ANI     X12  ; 下料旋臂旋轉垂直定點
      ANI     M210  ; 警報復歸
      OUT     T171 K100  ; 下料旋臂垂直異常延遲
211   LD      T171  ; 下料旋臂垂直異常延遲
      LD      M1688  ; 下料旋臂垂直異常
      ANI     M210  ; 警報復歸
      ORB
      OUT     M1688  ; 下料旋臂垂直異常
216   LD      M500  ; 下料旋臂水平SV
      LD      M220  ; 搬移啟動
      AND     X15  ; 下料旋臂長程下定點
      AND     X17  ; 下料旋臂短程下定點
      ANI     M500  ; 下料旋臂水平SV
      ANI     M501  ; 下料旋臂垂直SV
      ORB
      ANI     X10  ; 下料旋臂旋轉水平定點
      ANI     M210  ; 警報復歸
      OUT     T172 K100  ; 下料旋臂水平異常延遲
229   LD      T172  ; 下料旋臂水平異常延遲
      LD      M1689  ; 下料旋臂水平異常
      ANI     M210  ; 警報復歸
      ORB
      OUT     M1689  ; 下料旋臂水平異常
234   LDI     M1730  ; 出料空氣壓力異常
      MPS
      AND     Y107  ; 下料旋臂長程氣缸-上昇SV
      ANI     X13  ; 下料旋臂長程上定點
      OUT     T173 K100  ; 下料旋臂長程上異常延遲
      MPP
      AND     T173  ; 下料旋臂長程上異常延遲
      OUT     M1690  ; 下料旋臂長程上異常
245   LDI     M1730  ; 出料空氣壓力異常
      MPS
      AND     Y108  ; 下料旋臂長程氣缸-下降SV
      ANI     X15  ; 下料旋臂長程下定點
      OUT     T174 K100  ; 下料旋臂長程下異常延遲
      MPP
      AND     T174  ; 下料旋臂長程下異常延遲
      OUT     M1691  ; 下料旋臂長程下異常
256   LDI     M1730  ; 出料空氣壓力異常
      MPS
      AND     Y109  ; 下料旋臂短程氣缸-上昇SV
      ANI     X16  ; 下料旋臂短程上定點
      OUT     T175 K100  ; 下料旋臂短程上異常延遲
      MPP
      AND     T175  ; 下料旋臂短程上異常延遲
      OUT     M1692  ; 下料旋臂短程上異常
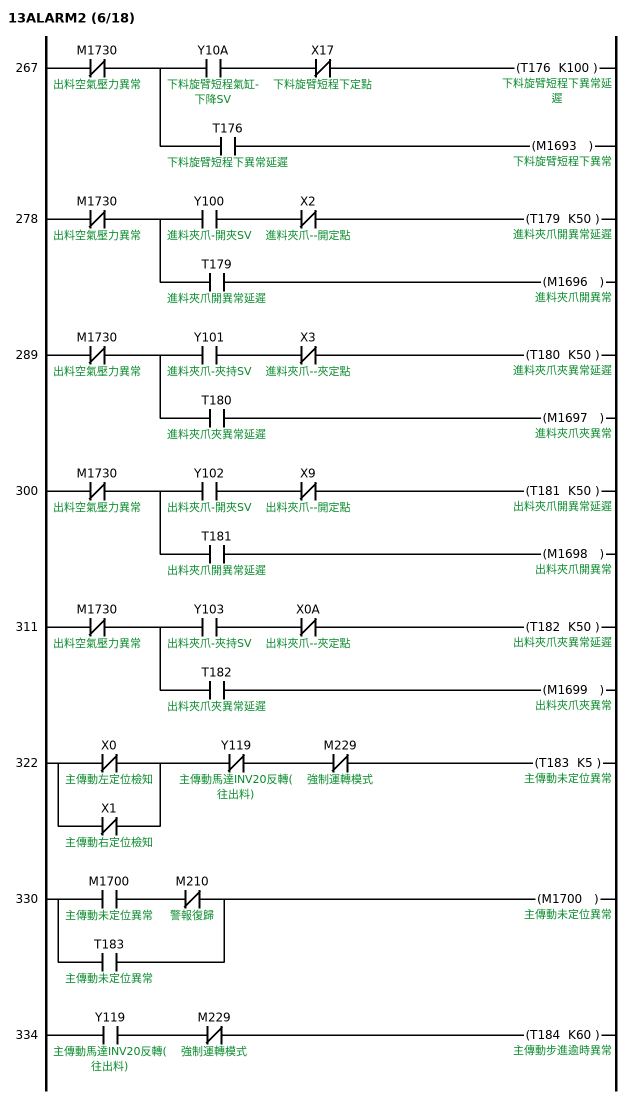
267   LDI     M1730  ; 出料空氣壓力異常
      MPS
      AND     Y10A  ; 下料旋臂短程氣缸-下降SV
      ANI     X17  ; 下料旋臂短程下定點
      OUT     T176 K100  ; 下料旋臂短程下異常延遲
      MPP
      AND     T176  ; 下料旋臂短程下異常延遲
      OUT     M1693  ; 下料旋臂短程下異常
278   LDI     M1730  ; 出料空氣壓力異常
      MPS
      AND     Y100  ; 進料夾爪-開夾SV
      ANI     X2  ; 進料夾爪--開定點
      OUT     T179 K50  ; 進料夾爪開異常延遲
      MPP
      AND     T179  ; 進料夾爪開異常延遲
      OUT     M1696  ; 進料夾爪開異常
289   LDI     M1730  ; 出料空氣壓力異常
      MPS
      AND     Y101  ; 進料夾爪-夾持SV
      ANI     X3  ; 進料夾爪--夾定點
      OUT     T180 K50  ; 進料夾爪夾異常延遲
      MPP
      AND     T180  ; 進料夾爪夾異常延遲
      OUT     M1697  ; 進料夾爪夾異常
300   LDI     M1730  ; 出料空氣壓力異常
      MPS
      AND     Y102  ; 出料夾爪-開夾SV
      ANI     X9  ; 出料夾爪--開定點
      OUT     T181 K50  ; 出料夾爪開異常延遲
      MPP
      AND     T181  ; 出料夾爪開異常延遲
      OUT     M1698  ; 出料夾爪開異常
311   LDI     M1730  ; 出料空氣壓力異常
      MPS
      AND     Y103  ; 出料夾爪-夾持SV
      ANI     X0A  ; 出料夾爪--夾定點
      OUT     T182 K50  ; 出料夾爪夾異常延遲
      MPP
      AND     T182  ; 出料夾爪夾異常延遲
      OUT     M1699  ; 出料夾爪夾異常
322   LDI     X0  ; 主傳動左定位檢知
      ORI     X1  ; 主傳動右定位檢知
      ANI     Y119  ; 主傳動馬達INV20反轉(往出料)
      ANI     M229  ; 強制運轉模式
      OUT     T183 K5  ; 主傳動未定位異常
330   LD      M1700  ; 主傳動未定位異常
      ANI     M210  ; 警報復歸
      OR      T183  ; 主傳動未定位異常
      OUT     M1700  ; 主傳動未定位異常
334   LD      Y119  ; 主傳動馬達INV20反轉(往出料)
      ANI     M229  ; 強制運轉模式
      OUT     T184 K60  ; 主傳動步進逾時異常
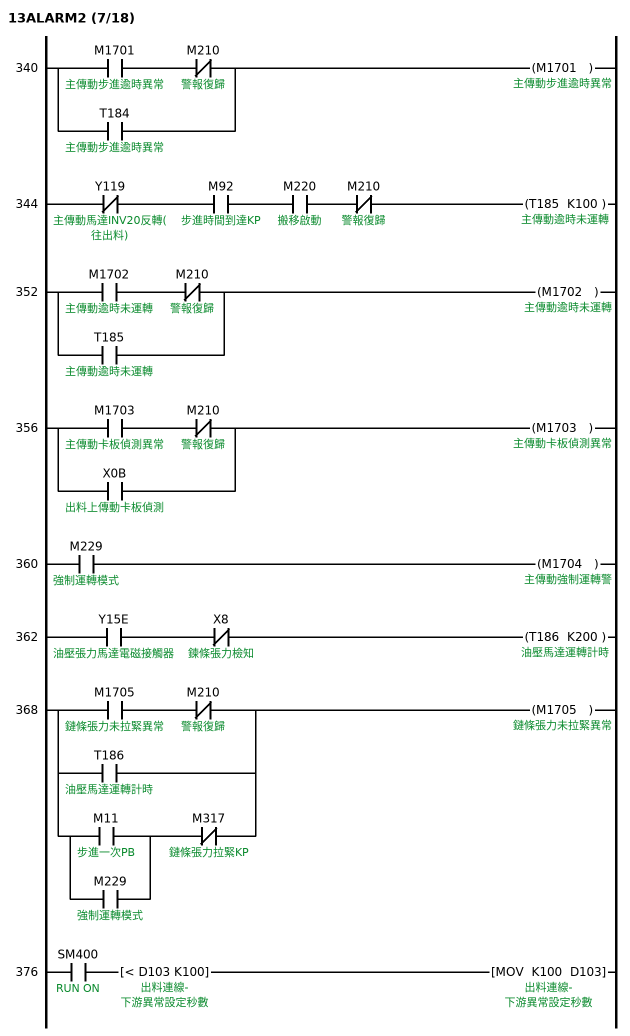
340   LD      M1701  ; 主傳動步進逾時異常
      ANI     M210  ; 警報復歸
      OR      T184  ; 主傳動步進逾時異常
      OUT     M1701  ; 主傳動步進逾時異常
344   LDI     Y119  ; 主傳動馬達INV20反轉(往出料)
      AND     M92  ; 步進時間到達KP
      AND     M220  ; 搬移啟動
      ANI     M210  ; 警報復歸
      OUT     T185 K100  ; 主傳動逾時未運轉
352   LD      M1702  ; 主傳動逾時未運轉
      ANI     M210  ; 警報復歸
      OR      T185  ; 主傳動逾時未運轉
      OUT     M1702  ; 主傳動逾時未運轉
356   LD      M1703  ; 主傳動卡板偵測異常
      ANI     M210  ; 警報復歸
      OR      X0B  ; 出料上傳動卡板偵測
      OUT     M1703  ; 主傳動卡板偵測異常
360   LD      M229  ; 強制運轉模式
      OUT     M1704  ; 主傳動強制運轉警
362   LD      Y15E  ; 油壓張力馬達電磁接觸器
      ANI     X8  ; 鍊條張力檢知
      OUT     T186 K200  ; 油壓馬達運轉計時
368   LD      M1705  ; 鏈條張力未拉緊異常
      ANI     M210  ; 警報復歸
      OR      T186  ; 油壓馬達運轉計時
      LD      M11  ; 步進一次PB
      OR      M229  ; 強制運轉模式
      ANI     M317  ; 鏈條張力拉緊KP
      ORB
      OUT     M1705  ; 鏈條張力未拉緊異常
376   LD      SM400  ; RUN ON
      AND<    D103 K100  ; 出料連線-下游異常設定秒數
      MOV     K100 D103
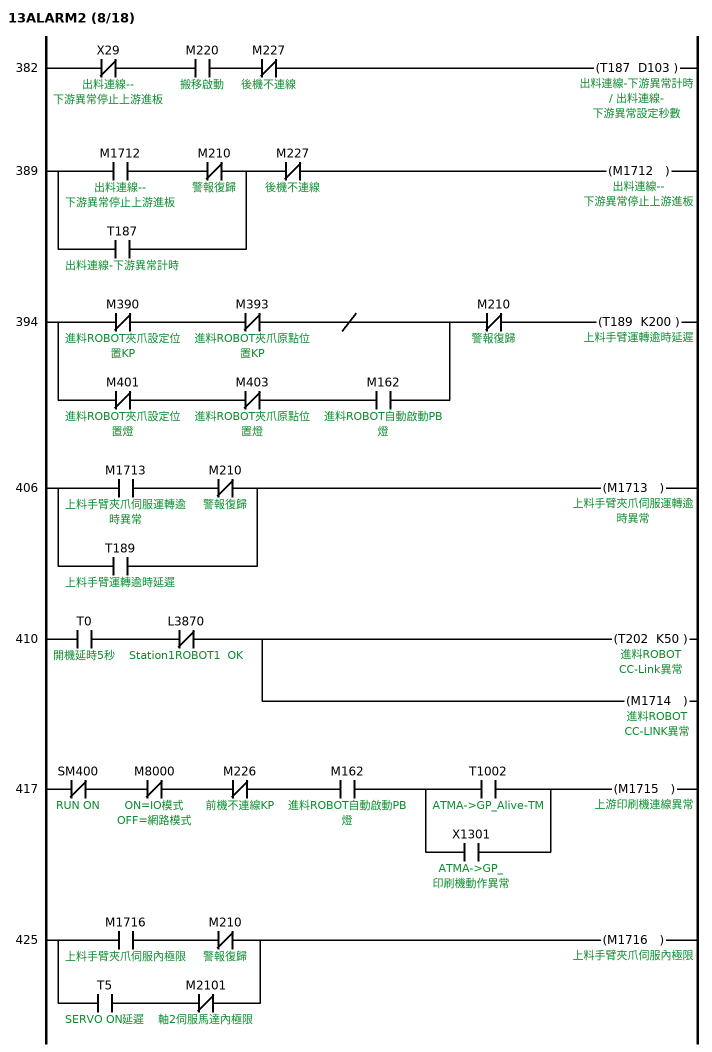
382   LDI     X29  ; 出料連線--下游異常停止上游進板
      AND     M220  ; 搬移啟動
      ANI     M227  ; 後機不連線
      OUT     T187 D103  ; 出料連線-下游異常計時 / 出料連線-下游異常設定秒數
389   LD      M1712  ; 出料連線--下游異常停止上游進板
      ANI     M210  ; 警報復歸
      OR      T187  ; 出料連線-下游異常計時
      ANI     M227  ; 後機不連線
      OUT     M1712  ; 出料連線--下游異常停止上游進板
394   LDI     M390  ; 進料ROBOT夾爪設定位置KP
      ANI     M393  ; 進料ROBOT夾爪原點位置KP
      INV
      LDI     M401  ; 進料ROBOT夾爪設定位置燈
      ANI     M403  ; 進料ROBOT夾爪原點位置燈
      AND     M162  ; 進料ROBOT自動啟動PB燈
      ORB
      ANI     M210  ; 警報復歸
      OUT     T189 K200  ; 上料手臂運轉逾時延遲
406   LD      M1713  ; 上料手臂夾爪伺服運轉逾時異常
      ANI     M210  ; 警報復歸
      OR      T189  ; 上料手臂運轉逾時延遲
      OUT     M1713  ; 上料手臂夾爪伺服運轉逾時異常
410   LD      T0  ; 開機延時5秒
      ANI     L3870  ; Station1ROBOT1  OK
      OUT     T202 K50  ; 進料ROBOT CC-Link異常
      OUT     M1714  ; 進料ROBOT CC-LINK異常
417   LDI     SM400  ; RUN ON
      ANI     M8000  ; ON=IO模式 OFF=網路模式
      ANI     M226  ; 前機不連線KP
      AND     M162  ; 進料ROBOT自動啟動PB燈
      LD      T1002  ; ATMA->GP_Alive-TM
      OR      X1301  ; ATMA->GP_印刷機動作異常
      ANB
      OUT     M1715  ; 上游印刷機連線異常
425   LD      M1716  ; 上料手臂夾爪伺服內極限
      ANI     M210  ; 警報復歸
      LD      T5  ; SERVO ON延遲
      ANI     M2101  ; 軸2伺服馬達內極限
      ORB
      OUT     M1716  ; 上料手臂夾爪伺服內極限
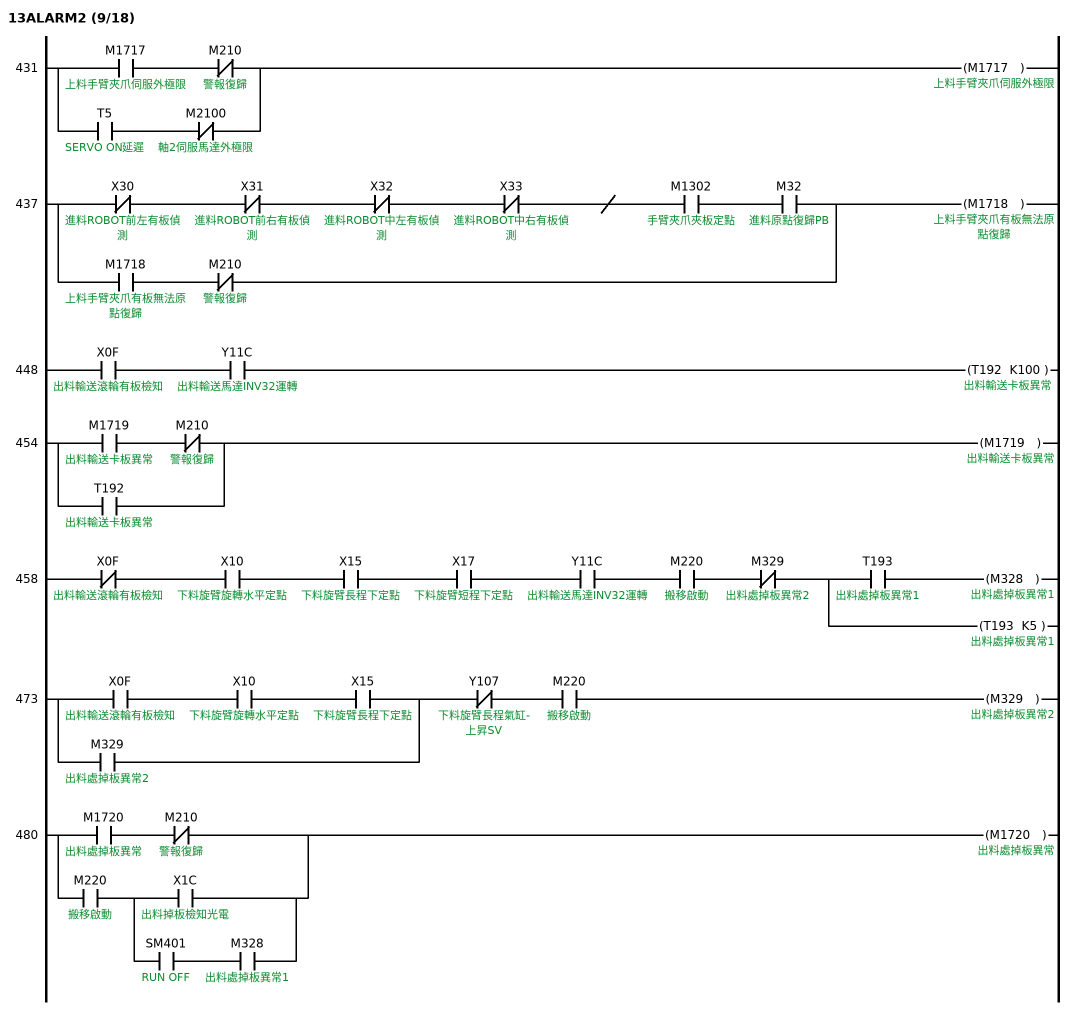
431   LD      M1717  ; 上料手臂夾爪伺服外極限
      ANI     M210  ; 警報復歸
      LD      T5  ; SERVO ON延遲
      ANI     M2100  ; 軸2伺服馬達外極限
      ORB
      OUT     M1717  ; 上料手臂夾爪伺服外極限
437   LDI     X30  ; 進料ROBOT前左有板偵測
      ANI     X31  ; 進料ROBOT前右有板偵測
      ANI     X32  ; 進料ROBOT中左有板偵測
      ANI     X33  ; 進料ROBOT中右有板偵測
      INV
      AND     M1302  ; 手臂夾爪夾板定點
      AND     M32  ; 進料原點復歸PB
      LD      M1718  ; 上料手臂夾爪有板無法原點復歸
      ANI     M210  ; 警報復歸
      ORB
      OUT     M1718  ; 上料手臂夾爪有板無法原點復歸
448   LD      X0F  ; 出料輸送滾輪有板檢知
      AND     Y11C  ; 出料輸送馬達INV32運轉
      OUT     T192 K100  ; 出料輸送卡板異常
454   LD      M1719  ; 出料輸送卡板異常
      ANI     M210  ; 警報復歸
      OR      T192  ; 出料輸送卡板異常
      OUT     M1719  ; 出料輸送卡板異常
458   LDI     X0F  ; 出料輸送滾輪有板檢知
      AND     X10  ; 下料旋臂旋轉水平定點
      AND     X15  ; 下料旋臂長程下定點
      AND     X17  ; 下料旋臂短程下定點
      AND     Y11C  ; 出料輸送馬達INV32運轉
      AND     M220  ; 搬移啟動
      ANI     M329  ; 出料處掉板異常2
      MPS
      AND     T193  ; 出料處掉板異常1
      OUT     M328  ; 出料處掉板異常1
      MPP
      OUT     T193 K5  ; 出料處掉板異常1
473   LD      X0F  ; 出料輸送滾輪有板檢知
      AND     X10  ; 下料旋臂旋轉水平定點
      AND     X15  ; 下料旋臂長程下定點
      OR      M329  ; 出料處掉板異常2
      ANI     Y107  ; 下料旋臂長程氣缸-上昇SV
      AND     M220  ; 搬移啟動
      OUT     M329  ; 出料處掉板異常2
480   LD      M1720  ; 出料處掉板異常
      ANI     M210  ; 警報復歸
      LD      M220  ; 搬移啟動
      LD      X1C  ; 出料掉板檢知光電
      LD      SM401  ; RUN OFF
      AND     M328  ; 出料處掉板異常1
      ORB
      ANB
      ORB
      OUT     M1720  ; 出料處掉板異常
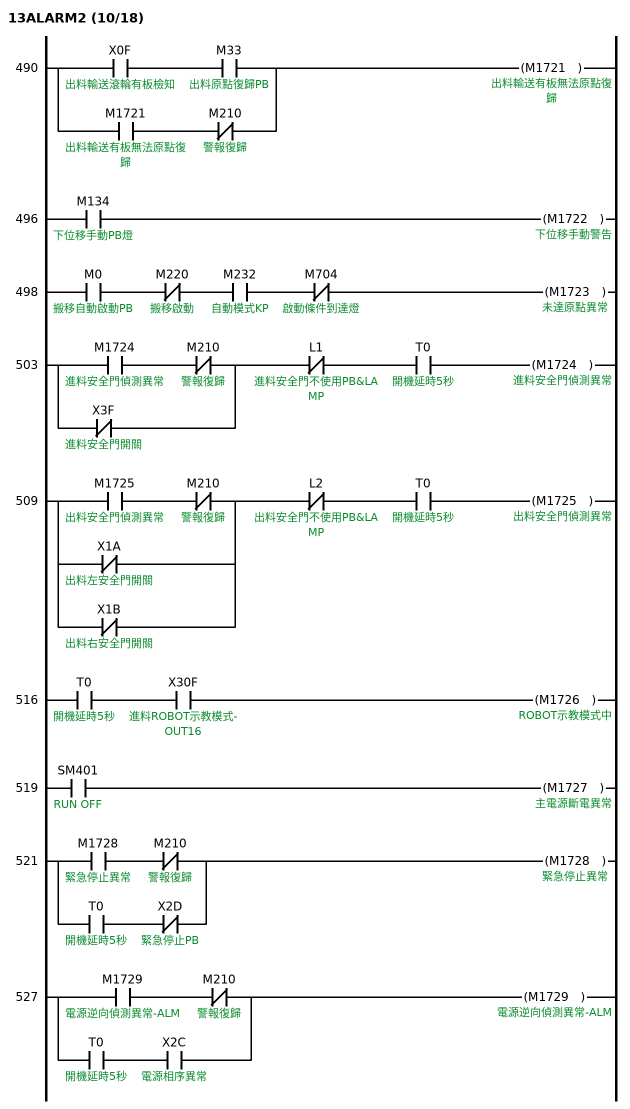
490   LD      X0F  ; 出料輸送滾輪有板檢知
      AND     M33  ; 出料原點復歸PB
      LD      M1721  ; 出料輸送有板無法原點復歸
      ANI     M210  ; 警報復歸
      ORB
      OUT     M1721  ; 出料輸送有板無法原點復歸
496   LD      M134  ; 下位移手動PB燈
      OUT     M1722  ; 下位移手動警告
498   LD      M0  ; 搬移自動啟動PB
      ANI     M220  ; 搬移啟動
      AND     M232  ; 自動模式KP
      ANI     M704  ; 啟動條件到達燈
      OUT     M1723  ; 未達原點異常
503   LD      M1724  ; 進料安全門偵測異常
      ANI     M210  ; 警報復歸
      ORI     X3F  ; 進料安全門開關
      ANI     L1  ; 進料安全門不使用PB&LAMP
      AND     T0  ; 開機延時5秒
      OUT     M1724  ; 進料安全門偵測異常
509   LD      M1725  ; 出料安全門偵測異常
      ANI     M210  ; 警報復歸
      ORI     X1A  ; 出料左安全門開關
      ORI     X1B  ; 出料右安全門開關
      ANI     L2  ; 出料安全門不使用PB&LAMP
      AND     T0  ; 開機延時5秒
      OUT     M1725  ; 出料安全門偵測異常
516   LD      T0  ; 開機延時5秒
      AND     X30F  ; 進料ROBOT示教模式-OUT16
      OUT     M1726  ; ROBOT示教模式中
519   LD      SM401  ; RUN OFF
      OUT     M1727  ; 主電源斷電異常
521   LD      M1728  ; 緊急停止異常
      ANI     M210  ; 警報復歸
      LD      T0  ; 開機延時5秒
      ANI     X2D  ; 緊急停止PB
      ORB
      OUT     M1728  ; 緊急停止異常
527   LD      M1729  ; 電源逆向偵測異常-ALM
      ANI     M210  ; 警報復歸
      LD      T0  ; 開機延時5秒
      AND     X2C  ; 電源相序異常
      ORB
      OUT     M1729  ; 電源逆向偵測異常-ALM
